TEXTLIST TextList_ISSstate
  0 = 'off'
  1 = 'initializing'
  2 = 'ready'
  100 = 'error'
   = ''
END_TEXTLIST

(* stored: Version 1.1.0.1, ProductVersion 3.1.4024.11
   TextList TextList_ISSstate: Id {c0563fe9-bd3d-40fe-86a1-661db7816ea7} *)
